% RSLogix 500 project Bag_Dryer_Fire_Jan_27_2022.RSS, saved by version 11.00.00.00 %
PROJECT "ML1200"    % processor: MicroLogix 1200; MAIN_PROG %

PROGRAM FILES
  LAD 2 "MAIN_PROG"  15 rungs
  LAD 3   11 rungs
  LAD 4   34 rungs
  LAD 5   12 rungs
  LAD 6   14 rungs
  LAD 7   2 rungs
  LAD 8   36 rungs
  LAD 9   2 rungs
  LAD 10   5 rungs
  LAD 11   14 rungs

DATA FILES
  O0 OUTPUT  8 elements
  I1 INPUT  19 elements
  S2 STATUS  66 elements
  B3 BINARY  20 elements
  T4 TIMER  11 elements
  C5 COUNTER  1 elements
  R6 CONTROL  1 elements
  N7 INTEGER  77 elements
  F8 FLOAT  1 elements
  PD9   3 elements

LADDER 2 "MAIN_PROG"
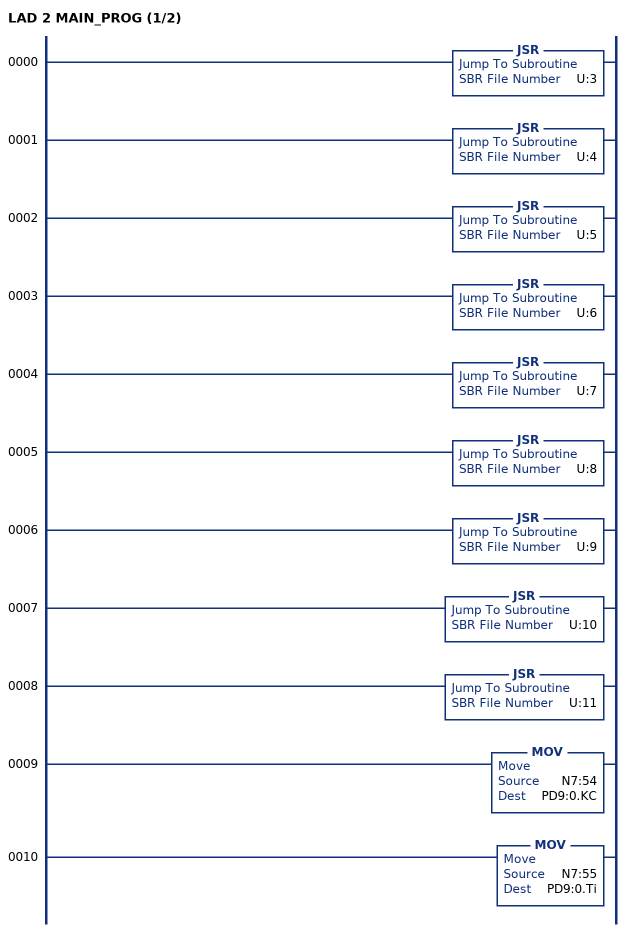
% Rung: 0 %
SOR JSR U:3 EOR
% Rung: 1 %
SOR JSR U:4 EOR
% Rung: 2 %
SOR JSR U:5 EOR
% Rung: 3 %
SOR JSR U:6 EOR
% Rung: 4 %
SOR JSR U:7 EOR
% Rung: 5 %
SOR JSR U:8 EOR
% Rung: 6 %
SOR JSR U:9 EOR
% Rung: 7 %
SOR JSR U:10 EOR
% Rung: 8 %
SOR JSR U:11 EOR
% Rung: 9 %
SOR MOV N7:54 PD9:0.KC EOR
% Rung: 10 %
SOR MOV N7:55 PD9:0.Ti EOR

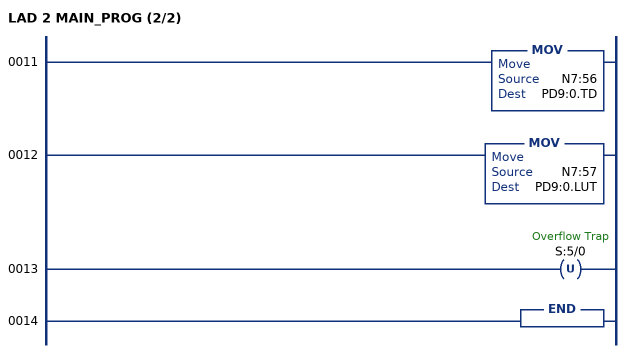
% Rung: 11 %
SOR MOV N7:56 PD9:0.TD EOR
% Rung: 12 %
SOR MOV N7:57 PD9:0.LUT EOR
% Rung: 13 %
SOR OTU S:5/0 EOR
%   S:5/0  "Overflow Trap" %
% Rung: 14 %
SOR END EOR

LADDER 3
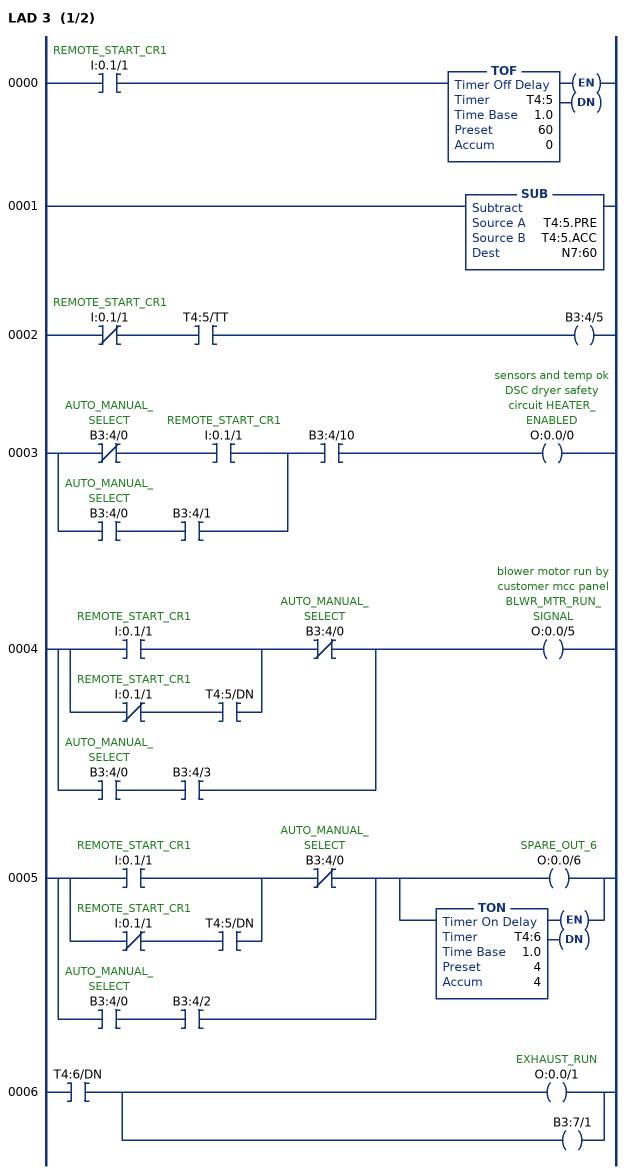
% Rung: 0 %
SOR XIC I:0.1/1 TOF T4:5 1.0 60 0 EOR
%   I:0.1/1  REMOTE_START_CR1 %
% Rung: 1 %
SOR SUB T4:5.PRE T4:5.ACC N7:60 EOR
% Rung: 2 %
SOR XIO I:0.1/1 XIC T4:5/TT OTE B3:4/5 EOR
%   I:0.1/1  REMOTE_START_CR1 %
% Rung: 3 %
SOR BST XIO B3:4/0 XIC I:0.1/1 NXB XIC B3:4/0 XIC B3:4/1 BND XIC B3:4/10 OTE O:0.0/0 EOR
%   B3:4/0  AUTO_MANUAL_SELECT %
%   I:0.1/1  REMOTE_START_CR1 %
%   O:0.0/0  HEATER_ENABLED  "sensors and temp ok DSC dryer safety circuit" %
% Rung: 4 %
SOR BST BST XIC I:0.1/1 NXB XIO I:0.1/1 XIC T4:5/DN BND XIO B3:4/0 NXB XIC B3:4/0 XIC B3:4/3 BND OTE O:0.0/5 EOR
%   I:0.1/1  REMOTE_START_CR1 %
%   B3:4/0  AUTO_MANUAL_SELECT %
%   O:0.0/5  BLWR_MTR_RUN_SIGNAL  "blower motor run by customer mcc panel" %
% Rung: 5 %
SOR BST BST XIC I:0.1/1 NXB XIO I:0.1/1 XIC T4:5/DN BND XIO B3:4/0 NXB XIC B3:4/0 XIC B3:4/2 BND BST OTE O:0.0/6 NXB TON T4:6 1.0 4 4 BND EOR
%   I:0.1/1  REMOTE_START_CR1 %
%   B3:4/0  AUTO_MANUAL_SELECT %
%   O:0.0/6  SPARE_OUT_6 %
% Rung: 6 %
SOR XIC T4:6/DN BST OTE O:0.0/1 NXB OTE B3:7/1 BND EOR
%   O:0.0/1  EXHAUST_RUN %

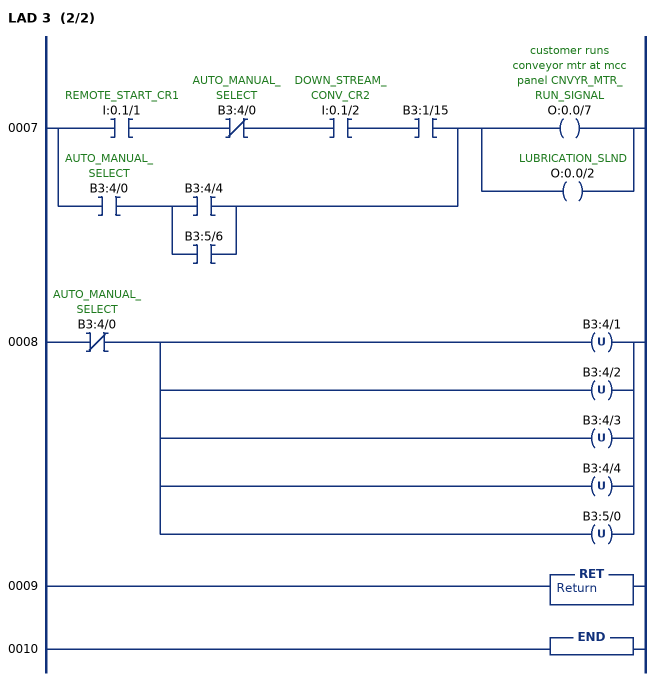
% Rung: 7 %
SOR BST XIC I:0.1/1 XIO B3:4/0 XIC I:0.1/2 XIC B3:1/15 NXB XIC B3:4/0 BST XIC B3:4/4 NXB XIC B3:5/6 BND BND BST OTE O:0.0/7 NXB OTE O:0.0/2 BND EOR
%   I:0.1/1  REMOTE_START_CR1 %
%   B3:4/0  AUTO_MANUAL_SELECT %
%   I:0.1/2  DOWN_STREAM_CONV_CR2 %
%   O:0.0/7  CNVYR_MTR_RUN_SIGNAL  "customer runs conveyor mtr at mcc panel" %
%   O:0.0/2  LUBRICATION_SLND %
% Rung: 8 %
SOR XIO B3:4/0 BST OTU B3:4/1 NXB BST OTU B3:4/2 NXB BST OTU B3:4/3 NXB BST OTU B3:4/4 NXB OTU B3:5/0 BND BND BND BND EOR
%   B3:4/0  AUTO_MANUAL_SELECT %
% Rung: 9 %
SOR RET EOR
% Rung: 10 %
SOR END EOR

LADDER 4
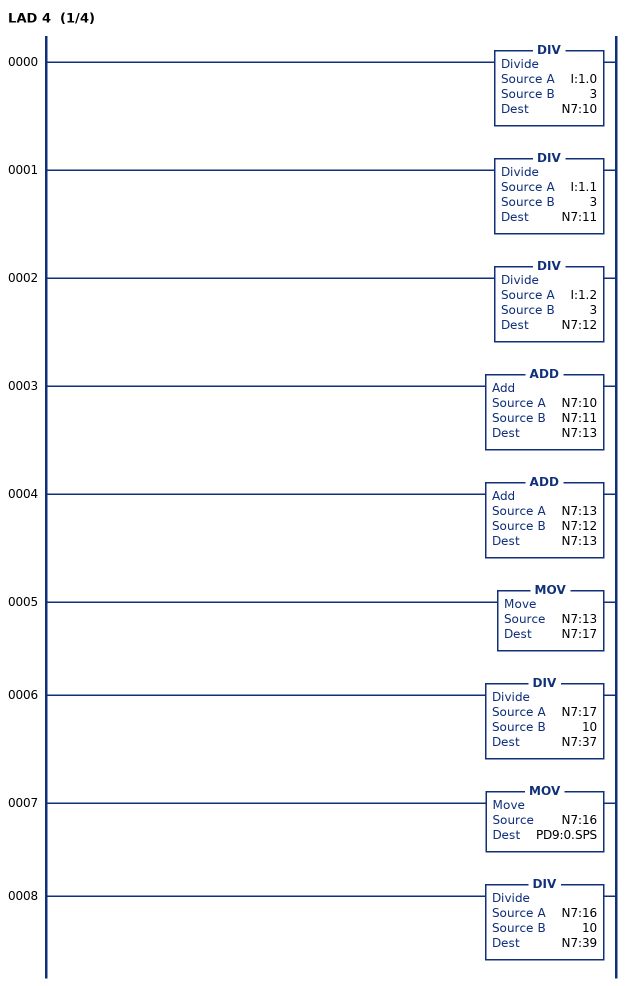
% Rung: 0 %
SOR DIV I:1.0 3 N7:10 EOR
% Rung: 1 %
SOR DIV I:1.1 3 N7:11 EOR
% Rung: 2 %
SOR DIV I:1.2 3 N7:12 EOR
% Rung: 3 %
SOR ADD N7:10 N7:11 N7:13 EOR
% Rung: 4 %
SOR ADD N7:13 N7:12 N7:13 EOR
% Rung: 5 %
SOR MOV N7:13 N7:17 EOR
% Rung: 6 %
SOR DIV N7:17 10 N7:37 EOR
% Rung: 7 %
SOR MOV N7:16 PD9:0.SPS EOR
% Rung: 8 %
SOR DIV N7:16 10 N7:39 EOR

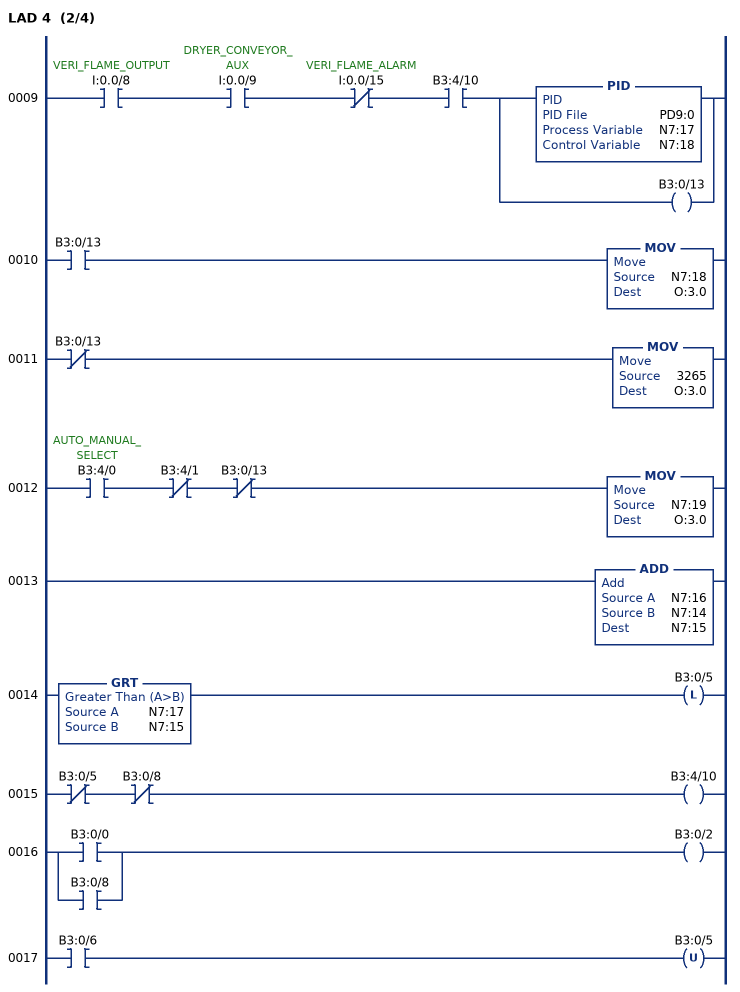
% Rung: 9 %
SOR XIC I:0.0/8 XIC I:0.0/9 XIO I:0.0/15 XIC B3:4/10 BST PID PD9:0 N7:17 N7:18 NXB OTE B3:0/13 BND EOR
%   I:0.0/8  VERI_FLAME_OUTPUT %
%   I:0.0/9  DRYER_CONVEYOR_AUX %
%   I:0.0/15  VERI_FLAME_ALARM %
% Rung: 10 %
SOR XIC B3:0/13 MOV N7:18 O:3.0 EOR
% Rung: 11 %
SOR XIO B3:0/13 MOV 3265 O:3.0 EOR
% Rung: 12 %
SOR XIC B3:4/0 XIO B3:4/1 XIO B3:0/13 MOV N7:19 O:3.0 EOR
%   B3:4/0  AUTO_MANUAL_SELECT %
% Rung: 13 %
SOR ADD N7:16 N7:14 N7:15 EOR
% Rung: 14 %
SOR GRT N7:17 N7:15 OTL B3:0/5 EOR
% Rung: 15 %
SOR XIO B3:0/5 XIO B3:0/8 OTE B3:4/10 EOR
% Rung: 16 %
SOR BST XIC B3:0/0 NXB XIC B3:0/8 BND OTE B3:0/2 EOR
% Rung: 17 %
SOR XIC B3:0/6 OTU B3:0/5 EOR

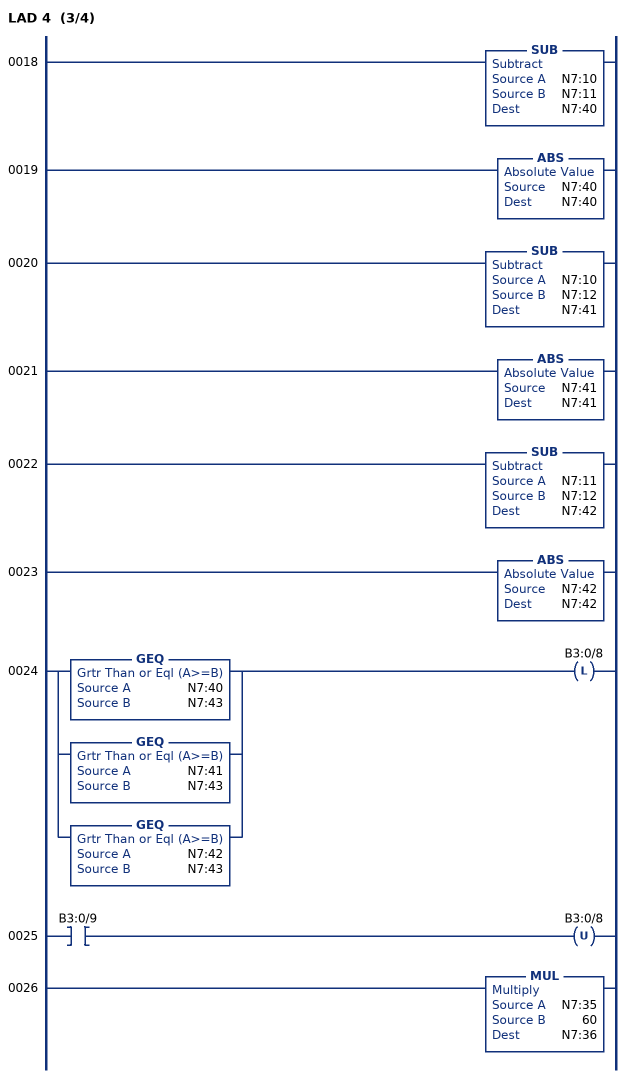
% Rung: 18 %
SOR SUB N7:10 N7:11 N7:40 EOR
% Rung: 19 %
SOR ABS N7:40 N7:40 EOR
% Rung: 20 %
SOR SUB N7:10 N7:12 N7:41 EOR
% Rung: 21 %
SOR ABS N7:41 N7:41 EOR
% Rung: 22 %
SOR SUB N7:11 N7:12 N7:42 EOR
% Rung: 23 %
SOR ABS N7:42 N7:42 EOR
% Rung: 24 %
SOR BST GEQ N7:40 N7:43 NXB BST GEQ N7:41 N7:43 NXB GEQ N7:42 N7:43 BND BND OTL B3:0/8 EOR
% Rung: 25 %
SOR XIC B3:0/9 OTU B3:0/8 EOR
% Rung: 26 %
SOR MUL N7:35 60 N7:36 EOR

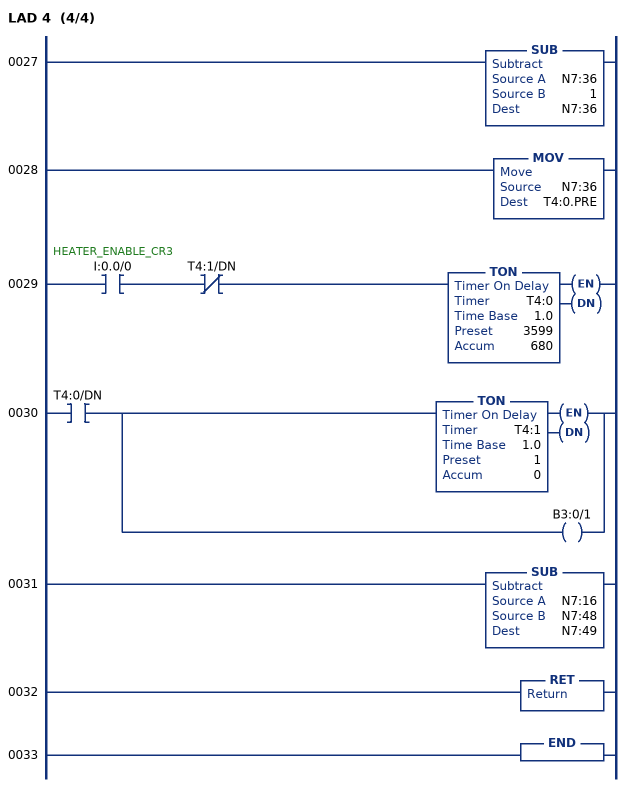
% Rung: 27 %
SOR SUB N7:36 1 N7:36 EOR
% Rung: 28 %
SOR MOV N7:36 T4:0.PRE EOR
% Rung: 29 %
SOR XIC I:0.0/0 XIO T4:1/DN TON T4:0 1.0 3599 680 EOR
%   I:0.0/0  HEATER_ENABLE_CR3 %
% Rung: 30 %
SOR XIC T4:0/DN BST TON T4:1 1.0 1 0 NXB OTE B3:0/1 BND EOR
% Rung: 31 %
SOR SUB N7:16 N7:48 N7:49 EOR
% Rung: 32 %
SOR RET EOR
% Rung: 33 %
SOR END EOR

LADDER 5
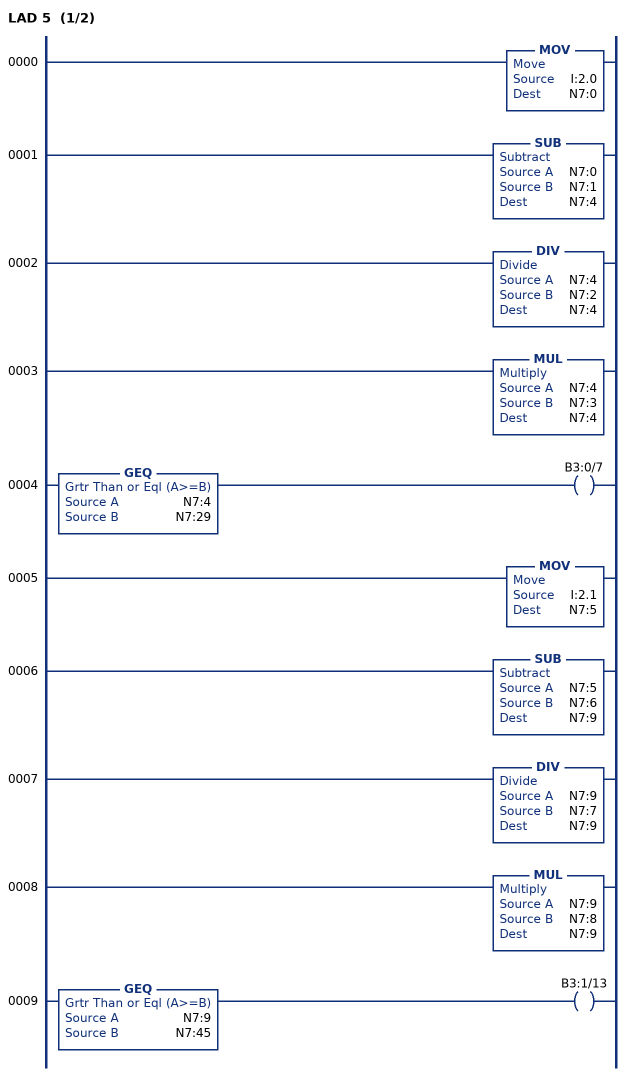
% Rung: 0 %
SOR MOV I:2.0 N7:0 EOR
% Rung: 1 %
SOR SUB N7:0 N7:1 N7:4 EOR
% Rung: 2 %
SOR DIV N7:4 N7:2 N7:4 EOR
% Rung: 3 %
SOR MUL N7:4 N7:3 N7:4 EOR
% Rung: 4 %
SOR GEQ N7:4 N7:29 OTE B3:0/7 EOR
% Rung: 5 %
SOR MOV I:2.1 N7:5 EOR
% Rung: 6 %
SOR SUB N7:5 N7:6 N7:9 EOR
% Rung: 7 %
SOR DIV N7:9 N7:7 N7:9 EOR
% Rung: 8 %
SOR MUL N7:9 N7:8 N7:9 EOR
% Rung: 9 %
SOR GEQ N7:9 N7:45 OTE B3:1/13 EOR

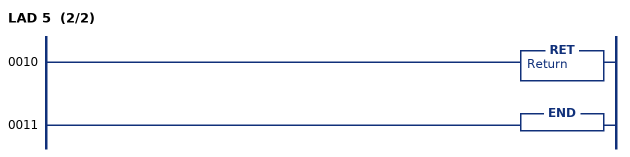
% Rung: 10 %
SOR RET EOR
% Rung: 11 %
SOR END EOR

LADDER 6
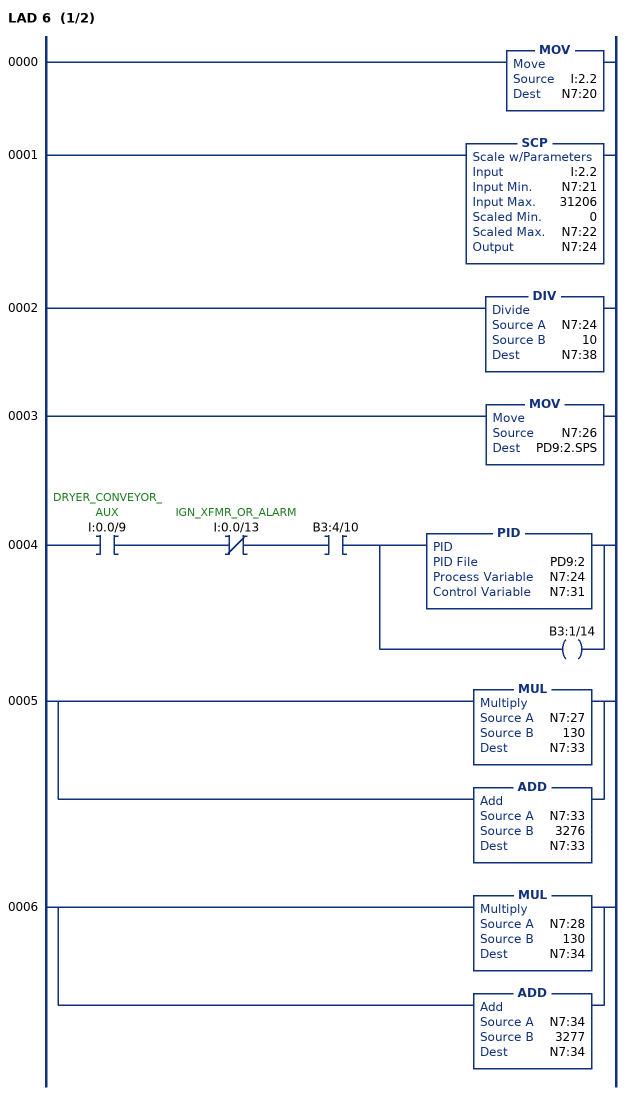
% Rung: 0 %
SOR MOV I:2.2 N7:20 EOR
% Rung: 1 %
SOR SCP I:2.2 N7:21 31206 0 N7:22 N7:24 EOR
% Rung: 2 %
SOR DIV N7:24 10 N7:38 EOR
% Rung: 3 %
SOR MOV N7:26 PD9:2.SPS EOR
% Rung: 4 %
SOR XIC I:0.0/9 XIO I:0.0/13 XIC B3:4/10 BST PID PD9:2 N7:24 N7:31 NXB OTE B3:1/14 BND EOR
%   I:0.0/9  DRYER_CONVEYOR_AUX %
%   I:0.0/13  IGN_XFMR_OR_ALARM %
% Rung: 5 %
SOR BST MUL N7:27 130 N7:33 NXB ADD N7:33 3276 N7:33 BND EOR
% Rung: 6 %
SOR BST MUL N7:28 130 N7:34 NXB ADD N7:34 3277 N7:34 BND EOR

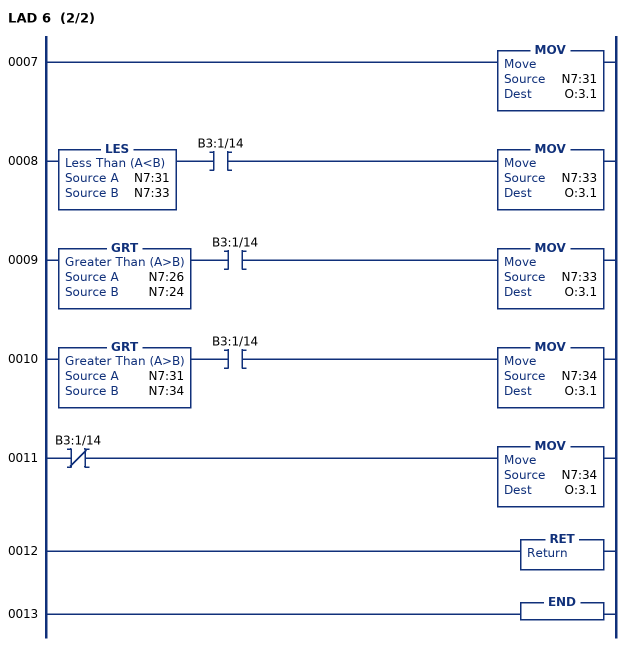
% Rung: 7 %
SOR MOV N7:31 O:3.1 EOR
% Rung: 8 %
SOR LES N7:31 N7:33 XIC B3:1/14 MOV N7:33 O:3.1 EOR
% Rung: 9 %
SOR GRT N7:26 N7:24 XIC B3:1/14 MOV N7:33 O:3.1 EOR
% Rung: 10 %
SOR GRT N7:31 N7:34 XIC B3:1/14 MOV N7:34 O:3.1 EOR
% Rung: 11 %
SOR XIO B3:1/14 MOV N7:34 O:3.1 EOR
% Rung: 12 %
SOR RET EOR
% Rung: 13 %
SOR END EOR

LADDER 7
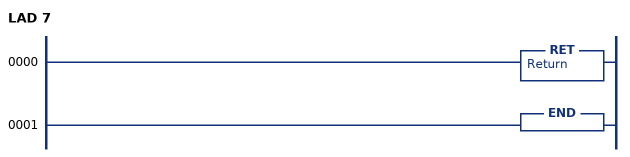
% Rung: 0 %
SOR RET EOR
% Rung: 1 %
SOR END EOR

LADDER 8
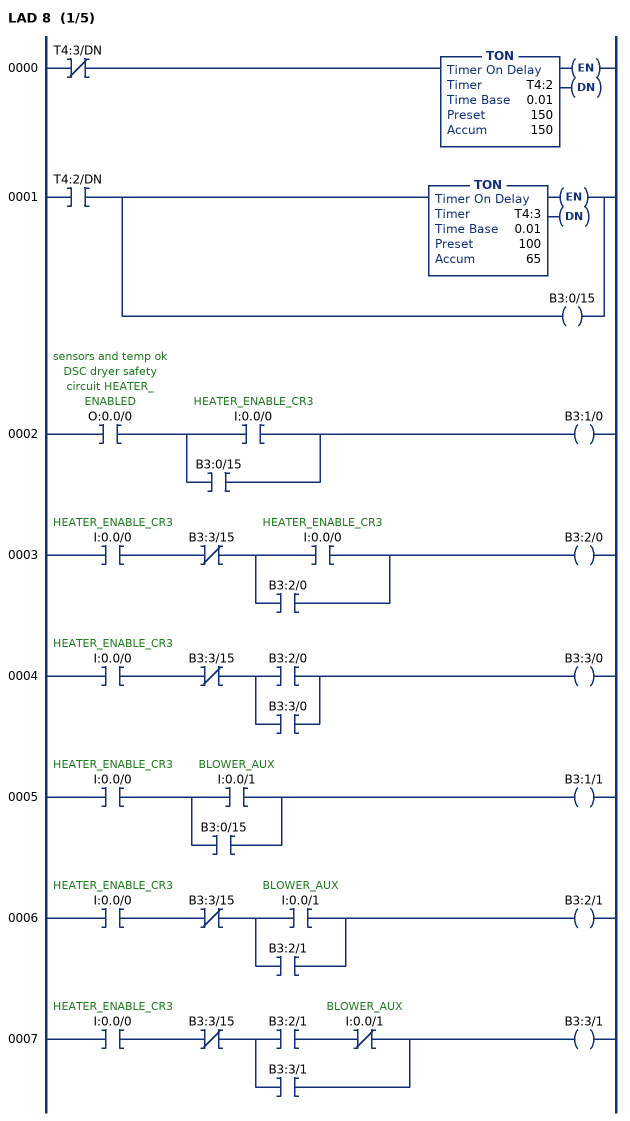
% Rung: 0 %
SOR XIO T4:3/DN TON T4:2 0.01 150 150 EOR
% Rung: 1 %
SOR XIC T4:2/DN BST TON T4:3 0.01 100 65 NXB OTE B3:0/15 BND EOR
% Rung: 2 %
SOR XIC O:0.0/0 BST XIC I:0.0/0 NXB XIC B3:0/15 BND OTE B3:1/0 EOR
%   O:0.0/0  HEATER_ENABLED  "sensors and temp ok DSC dryer safety circuit" %
%   I:0.0/0  HEATER_ENABLE_CR3 %
% Rung: 3 %
SOR XIC I:0.0/0 XIO B3:3/15 BST XIC I:0.0/0 NXB XIC B3:2/0 BND OTE B3:2/0 EOR
%   I:0.0/0  HEATER_ENABLE_CR3 %
% Rung: 4 %
SOR XIC I:0.0/0 XIO B3:3/15 BST XIC B3:2/0 NXB XIC B3:3/0 BND OTE B3:3/0 EOR
%   I:0.0/0  HEATER_ENABLE_CR3 %
% Rung: 5 %
SOR XIC I:0.0/0 BST XIC I:0.0/1 NXB XIC B3:0/15 BND OTE B3:1/1 EOR
%   I:0.0/0  HEATER_ENABLE_CR3 %
%   I:0.0/1  BLOWER_AUX %
% Rung: 6 %
SOR XIC I:0.0/0 XIO B3:3/15 BST XIC I:0.0/1 NXB XIC B3:2/1 BND OTE B3:2/1 EOR
%   I:0.0/0  HEATER_ENABLE_CR3 %
%   I:0.0/1  BLOWER_AUX %
% Rung: 7 %
SOR XIC I:0.0/0 XIO B3:3/15 BST XIC B3:2/1 XIO I:0.0/1 NXB XIC B3:3/1 BND OTE B3:3/1 EOR
%   I:0.0/0  HEATER_ENABLE_CR3 %
%   I:0.0/1  BLOWER_AUX %

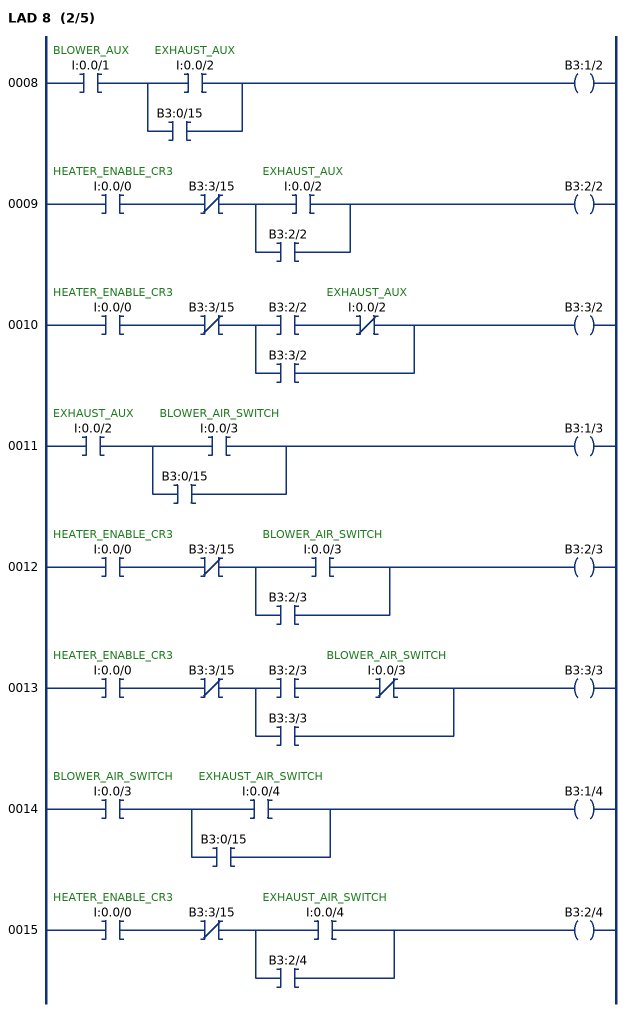
% Rung: 8 %
SOR XIC I:0.0/1 BST XIC I:0.0/2 NXB XIC B3:0/15 BND OTE B3:1/2 EOR
%   I:0.0/1  BLOWER_AUX %
%   I:0.0/2  EXHAUST_AUX %
% Rung: 9 %
SOR XIC I:0.0/0 XIO B3:3/15 BST XIC I:0.0/2 NXB XIC B3:2/2 BND OTE B3:2/2 EOR
%   I:0.0/0  HEATER_ENABLE_CR3 %
%   I:0.0/2  EXHAUST_AUX %
% Rung: 10 %
SOR XIC I:0.0/0 XIO B3:3/15 BST XIC B3:2/2 XIO I:0.0/2 NXB XIC B3:3/2 BND OTE B3:3/2 EOR
%   I:0.0/0  HEATER_ENABLE_CR3 %
%   I:0.0/2  EXHAUST_AUX %
% Rung: 11 %
SOR XIC I:0.0/2 BST XIC I:0.0/3 NXB XIC B3:0/15 BND OTE B3:1/3 EOR
%   I:0.0/2  EXHAUST_AUX %
%   I:0.0/3  BLOWER_AIR_SWITCH %
% Rung: 12 %
SOR XIC I:0.0/0 XIO B3:3/15 BST XIC I:0.0/3 NXB XIC B3:2/3 BND OTE B3:2/3 EOR
%   I:0.0/0  HEATER_ENABLE_CR3 %
%   I:0.0/3  BLOWER_AIR_SWITCH %
% Rung: 13 %
SOR XIC I:0.0/0 XIO B3:3/15 BST XIC B3:2/3 XIO I:0.0/3 NXB XIC B3:3/3 BND OTE B3:3/3 EOR
%   I:0.0/0  HEATER_ENABLE_CR3 %
%   I:0.0/3  BLOWER_AIR_SWITCH %
% Rung: 14 %
SOR XIC I:0.0/3 BST XIC I:0.0/4 NXB XIC B3:0/15 BND OTE B3:1/4 EOR
%   I:0.0/3  BLOWER_AIR_SWITCH %
%   I:0.0/4  EXHAUST_AIR_SWITCH %
% Rung: 15 %
SOR XIC I:0.0/0 XIO B3:3/15 BST XIC I:0.0/4 NXB XIC B3:2/4 BND OTE B3:2/4 EOR
%   I:0.0/0  HEATER_ENABLE_CR3 %
%   I:0.0/4  EXHAUST_AIR_SWITCH %

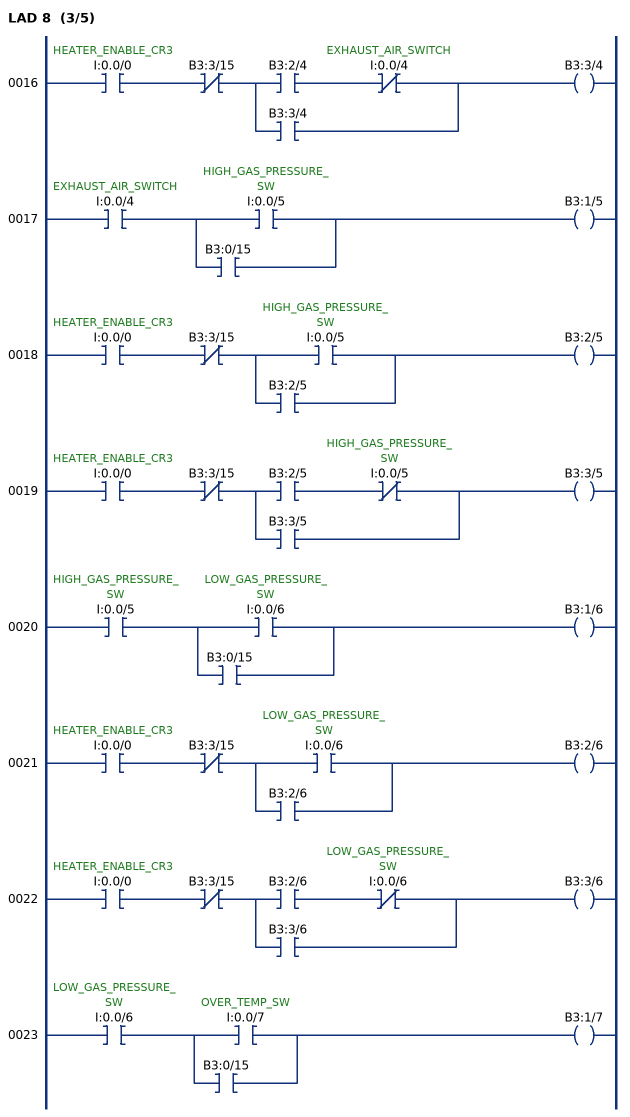
% Rung: 16 %
SOR XIC I:0.0/0 XIO B3:3/15 BST XIC B3:2/4 XIO I:0.0/4 NXB XIC B3:3/4 BND OTE B3:3/4 EOR
%   I:0.0/0  HEATER_ENABLE_CR3 %
%   I:0.0/4  EXHAUST_AIR_SWITCH %
% Rung: 17 %
SOR XIC I:0.0/4 BST XIC I:0.0/5 NXB XIC B3:0/15 BND OTE B3:1/5 EOR
%   I:0.0/4  EXHAUST_AIR_SWITCH %
%   I:0.0/5  HIGH_GAS_PRESSURE_SW %
% Rung: 18 %
SOR XIC I:0.0/0 XIO B3:3/15 BST XIC I:0.0/5 NXB XIC B3:2/5 BND OTE B3:2/5 EOR
%   I:0.0/0  HEATER_ENABLE_CR3 %
%   I:0.0/5  HIGH_GAS_PRESSURE_SW %
% Rung: 19 %
SOR XIC I:0.0/0 XIO B3:3/15 BST XIC B3:2/5 XIO I:0.0/5 NXB XIC B3:3/5 BND OTE B3:3/5 EOR
%   I:0.0/0  HEATER_ENABLE_CR3 %
%   I:0.0/5  HIGH_GAS_PRESSURE_SW %
% Rung: 20 %
SOR XIC I:0.0/5 BST XIC I:0.0/6 NXB XIC B3:0/15 BND OTE B3:1/6 EOR
%   I:0.0/5  HIGH_GAS_PRESSURE_SW %
%   I:0.0/6  LOW_GAS_PRESSURE_SW %
% Rung: 21 %
SOR XIC I:0.0/0 XIO B3:3/15 BST XIC I:0.0/6 NXB XIC B3:2/6 BND OTE B3:2/6 EOR
%   I:0.0/0  HEATER_ENABLE_CR3 %
%   I:0.0/6  LOW_GAS_PRESSURE_SW %
% Rung: 22 %
SOR XIC I:0.0/0 XIO B3:3/15 BST XIC B3:2/6 XIO I:0.0/6 NXB XIC B3:3/6 BND OTE B3:3/6 EOR
%   I:0.0/0  HEATER_ENABLE_CR3 %
%   I:0.0/6  LOW_GAS_PRESSURE_SW %
% Rung: 23 %
SOR XIC I:0.0/6 BST XIC I:0.0/7 NXB XIC B3:0/15 BND OTE B3:1/7 EOR
%   I:0.0/6  LOW_GAS_PRESSURE_SW %
%   I:0.0/7  OVER_TEMP_SW %

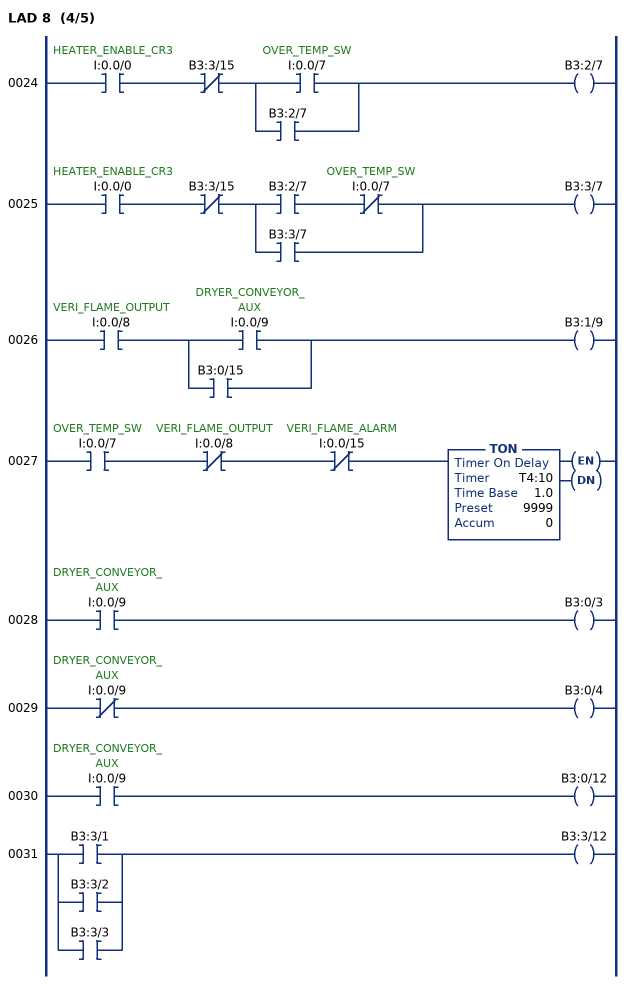
% Rung: 24 %
SOR XIC I:0.0/0 XIO B3:3/15 BST XIC I:0.0/7 NXB XIC B3:2/7 BND OTE B3:2/7 EOR
%   I:0.0/0  HEATER_ENABLE_CR3 %
%   I:0.0/7  OVER_TEMP_SW %
% Rung: 25 %
SOR XIC I:0.0/0 XIO B3:3/15 BST XIC B3:2/7 XIO I:0.0/7 NXB XIC B3:3/7 BND OTE B3:3/7 EOR
%   I:0.0/0  HEATER_ENABLE_CR3 %
%   I:0.0/7  OVER_TEMP_SW %
% Rung: 26 %
SOR XIC I:0.0/8 BST XIC I:0.0/9 NXB XIC B3:0/15 BND OTE B3:1/9 EOR
%   I:0.0/8  VERI_FLAME_OUTPUT %
%   I:0.0/9  DRYER_CONVEYOR_AUX %
% Rung: 27 %
SOR XIC I:0.0/7 XIO I:0.0/8 XIO I:0.0/15 TON T4:10 1.0 9999 0 EOR
%   I:0.0/7  OVER_TEMP_SW %
%   I:0.0/8  VERI_FLAME_OUTPUT %
%   I:0.0/15  VERI_FLAME_ALARM %
% Rung: 28 %
SOR XIC I:0.0/9 OTE B3:0/3 EOR
%   I:0.0/9  DRYER_CONVEYOR_AUX %
% Rung: 29 %
SOR XIO I:0.0/9 OTE B3:0/4 EOR
%   I:0.0/9  DRYER_CONVEYOR_AUX %
% Rung: 30 %
SOR XIC I:0.0/9 OTE B3:0/12 EOR
%   I:0.0/9  DRYER_CONVEYOR_AUX %
% Rung: 31 %
SOR BST XIC B3:3/1 NXB BST XIC B3:3/2 NXB XIC B3:3/3 BND BND OTE B3:3/12 EOR

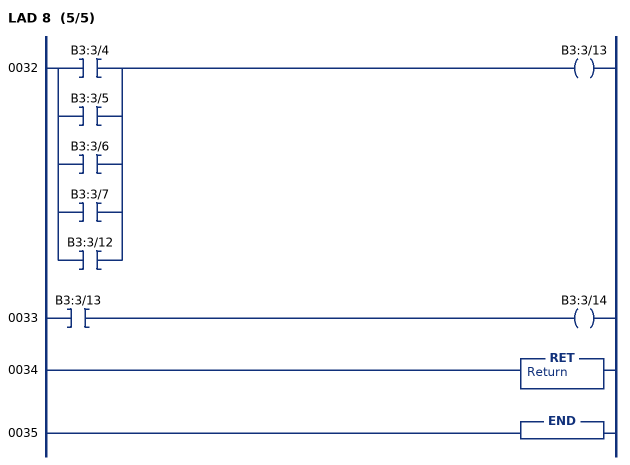
% Rung: 32 %
SOR BST XIC B3:3/4 NXB BST XIC B3:3/5 NXB BST XIC B3:3/6 NXB BST XIC B3:3/7 NXB XIC B3:3/12 BND BND BND BND OTE B3:3/13 EOR
% Rung: 33 %
SOR XIC B3:3/13 OTE B3:3/14 EOR
% Rung: 34 %
SOR RET EOR
% Rung: 35 %
SOR END EOR

LADDER 9
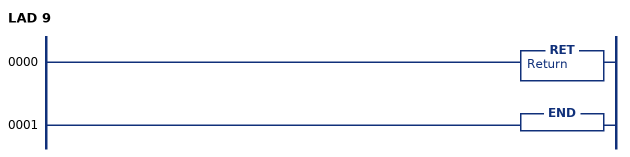
% Rung: 0 %
SOR RET EOR
% Rung: 1 %
SOR END EOR

LADDER 10
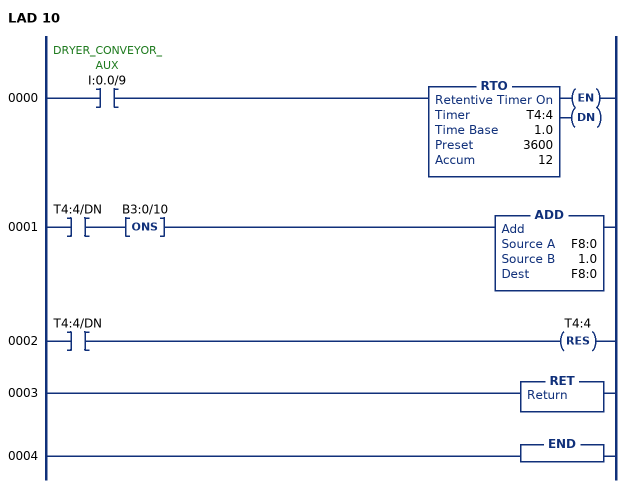
% Rung: 0 %
SOR XIC I:0.0/9 RTO T4:4 1.0 3600 12 EOR
%   I:0.0/9  DRYER_CONVEYOR_AUX %
% Rung: 1 %
SOR XIC T4:4/DN ONS B3:0/10 ADD F8:0 1.0 F8:0 EOR
% Rung: 2 %
SOR XIC T4:4/DN RES T4:4 EOR
% Rung: 3 %
SOR RET EOR
% Rung: 4 %
SOR END EOR

LADDER 11
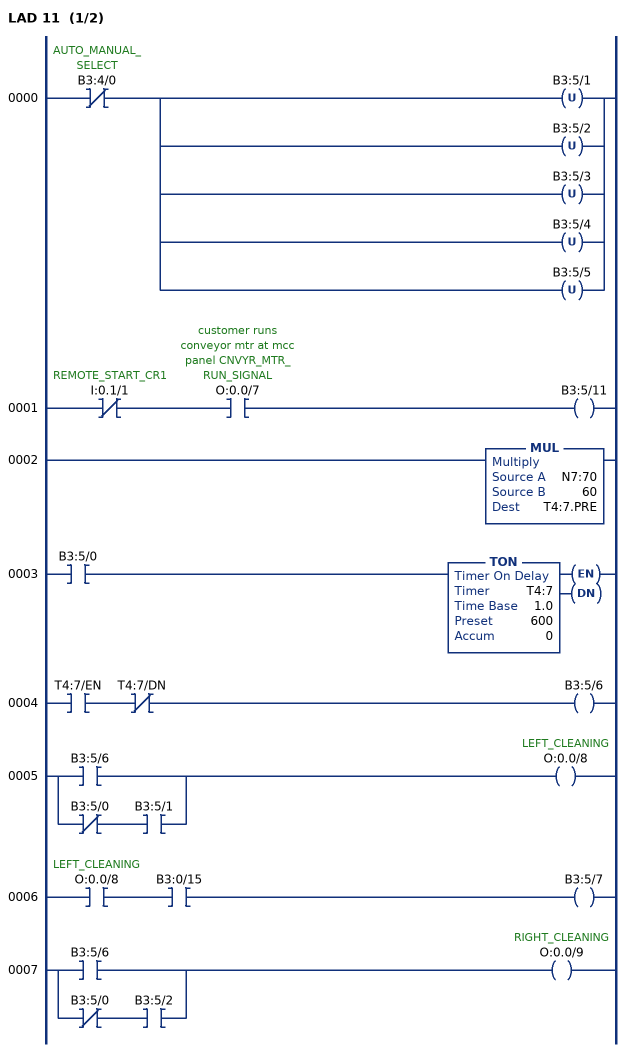
% Rung: 0 %
SOR XIO B3:4/0 BST OTU B3:5/1 NXB BST OTU B3:5/2 NXB BST OTU B3:5/3 NXB BST OTU B3:5/4 NXB OTU B3:5/5 BND BND BND BND EOR
%   B3:4/0  AUTO_MANUAL_SELECT %
% Rung: 1 %
SOR XIO I:0.1/1 XIC O:0.0/7 OTE B3:5/11 EOR
%   I:0.1/1  REMOTE_START_CR1 %
%   O:0.0/7  CNVYR_MTR_RUN_SIGNAL  "customer runs conveyor mtr at mcc panel" %
% Rung: 2 %
SOR MUL N7:70 60 T4:7.PRE EOR
% Rung: 3 %
SOR XIC B3:5/0 TON T4:7 1.0 600 0 EOR
% Rung: 4 %
SOR XIC T4:7/EN XIO T4:7/DN OTE B3:5/6 EOR
% Rung: 5 %
SOR BST XIC B3:5/6 NXB XIO B3:5/0 XIC B3:5/1 BND OTE O:0.0/8 EOR
%   O:0.0/8  LEFT_CLEANING %
% Rung: 6 %
SOR XIC O:0.0/8 XIC B3:0/15 OTE B3:5/7 EOR
%   O:0.0/8  LEFT_CLEANING %
% Rung: 7 %
SOR BST XIC B3:5/6 NXB XIO B3:5/0 XIC B3:5/2 BND OTE O:0.0/9 EOR
%   O:0.0/9  RIGHT_CLEANING %

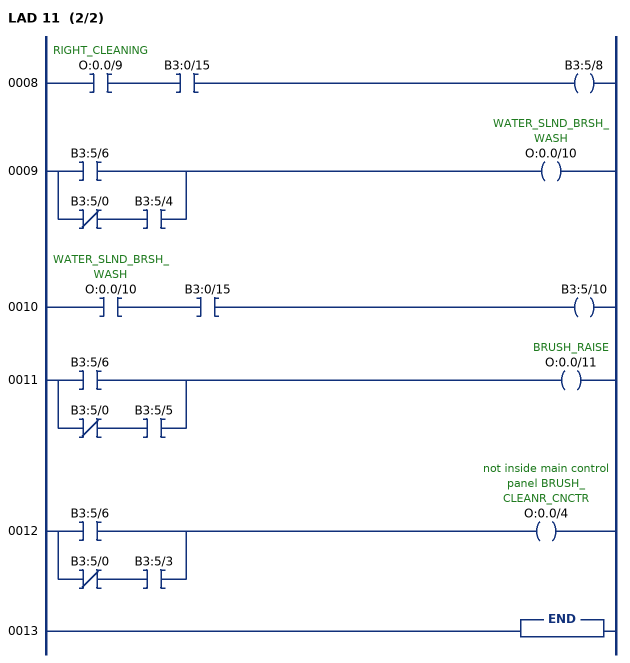
% Rung: 8 %
SOR XIC O:0.0/9 XIC B3:0/15 OTE B3:5/8 EOR
%   O:0.0/9  RIGHT_CLEANING %
% Rung: 9 %
SOR BST XIC B3:5/6 NXB XIO B3:5/0 XIC B3:5/4 BND OTE O:0.0/10 EOR
%   O:0.0/10  WATER_SLND_BRSH_WASH %
% Rung: 10 %
SOR XIC O:0.0/10 XIC B3:0/15 OTE B3:5/10 EOR
%   O:0.0/10  WATER_SLND_BRSH_WASH %
% Rung: 11 %
SOR BST XIC B3:5/6 NXB XIO B3:5/0 XIC B3:5/5 BND OTE O:0.0/11 EOR
%   O:0.0/11  BRUSH_RAISE %
% Rung: 12 %
SOR BST XIC B3:5/6 NXB XIO B3:5/0 XIC B3:5/3 BND OTE O:0.0/4 EOR
%   O:0.0/4  BRUSH_CLEANR_CNCTR  "not inside main control panel" %
% Rung: 13 %
SOR END EOR

OTHER DOCUMENTED ADDRESSES
  I:0.0/10  SPARE_10
  I:0.0/11  PILOT_GAS_VALVE
  I:0.0/12  SPARE_12
  I:0.0/14  SPARE_14
  I:0.1/0  SPARE_16
  O:0.0/3  SPARE_OUT_3

DATA TABLE (non-zero values as saved)
DATA B3
% B3:0 % 0XB008 0XC2FF 0X00FF 0X0001 0X0580 0X0000 0X0000 0X0102 0X0000 0X0000
% B3:10 % 0X0001 0X0000 0X0000 0X0000 0X0000 0X0000 0X0000 0X0000 0X0000 0X0000
DATA T4
% .PRE .ACC %
% T4:0 % 3599 680
% T4:1 % 1 0
% T4:2 % 150 150
% T4:3 % 100 65
% T4:4 % 3600 12
% T4:5 % 60 0
% T4:6 % 4 4
% T4:7 % 600 0
% T4:8 % 600 0
% T4:9 % 1800 0
% T4:10 % 9999 0
DATA N7
% N7:0 % 7684 6226 105 1 14 6280 6265 18 1 1
% N7:10 % 371 367 374 1112 200 1300 1100 1112 7888 3265
% N7:20 % 11558 6250 1000 10 213 25 25 75 100 15
% N7:30 % 10 0 195 13026 16277 60 3599 111 21 110
% N7:40 % 4 3 7 200 0 5 0 0 0 1100
% N7:50 % 0 10 0 0 60 2 20 300 0 0
% N7:60 % 60 0 0 0 0 0 0 0 0 0
% N7:70 % 10 0 0 0 0 0 0
DATA F8
% F8:0 % 404
